# EPICS autosave request: iocBoot/sioc-esb-ct01/ct01.req
$(P):NCOUNTS
$(P):THRESH
